// Mitsubishi GX Works2 project: DZRN_home   PLC: FX3U/FX3UC

PROGRAM MAIN
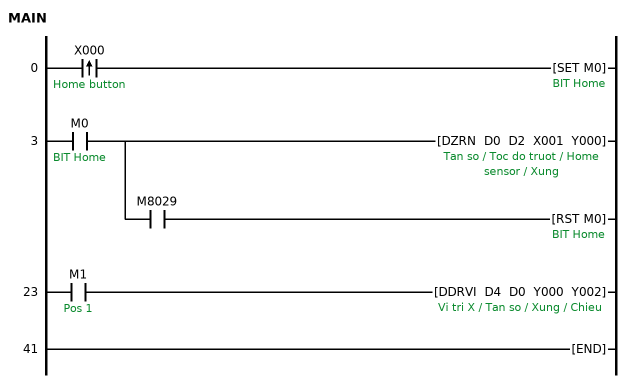
0     LDP     X000  ; Home button
      SET     M0  ; BIT Home
3     LD      M0  ; BIT Home
      DZRN    D0 D2 X001 Y000  ; Tan so / Toc do truot / Home sensor / Xung
      AND     M8029
      RST     M0  ; BIT Home
23    LD      M1  ; Pos 1
      DDRVI   D4 D0 Y000 Y002  ; Vi tri X / Chieu
41    END
END_PROGRAM

// device comments not shown above
M2  ; Pos 2
M3  ; Pos 3
